(* Logix 5000 project; controller AMANA_DC_PLANT_01 vendor 1 type 14 code 164 rev 31.12; software revision 31.02; part 9 of 9 *)
(* tags used below, declared in another part *)
   Barcode_Longest : DINT;
   Barcode_Shortest : DINT;
   Comma : STRING;
   Counters : COUNTER[16];
   MSG_Enable : DINT;
   MSG_ONS : DINT;
   MSG_Steps : DINT;
   NULL_String : STRING;
   SCANNER_DOCKSORTING_DATA : Keyence_2_Barcode;
   Timer_MSG_Interval : TIMER;
   Read_From_Clearpack_1 : MESSAGE;
   Read_From_L4_1 : MESSAGE;
   Read_From_L6_1 : MESSAGE;
   Read_From_L7_1 : MESSAGE;
   Read_From_Merge_1 : MESSAGE;
   Read_From_Sort_1 : MESSAGE;
(* OH_BARCODE_SCAN, continued *)

ROUTINE R11_DOCKSORTING   (* ladder *)
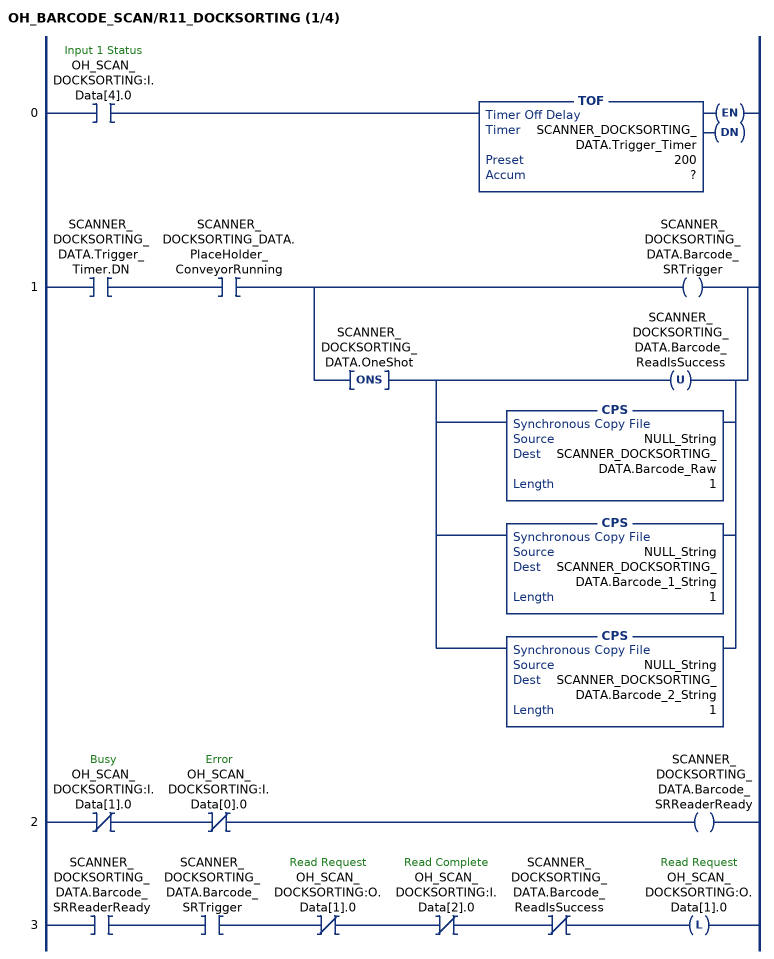
   0: XIC(OH_SCAN_DOCKSORTING:I.Data[4].0)TOF(SCANNER_DOCKSORTING_DATA.Trigger_Timer,?,?);
   1: XIC(SCANNER_DOCKSORTING_DATA.Trigger_Timer.DN)XIC(SCANNER_DOCKSORTING_DATA.PlaceHolder_ConveyorRunning)[OTE(SCANNER_DOCKSORTING_DATA.Barcode_SRTrigger) ,ONS(SCANNER_DOCKSORTING_DATA.OneShot) [OTU(SCANNER_DOCKSORTING_DATA.Barcode_ReadIsSuccess) ,CPS(NULL_String,SCANNER_DOCKSORTING_DATA.Barcode_Raw,1) ,CPS(NULL_String,SCANNER_DOCKSORTING_DATA.Barcode_1_String,1) ,CPS(NULL_String,SCANNER_DOCKSORTING_DATA.Barcode_2_String,1) ] ];
   2: XIO(OH_SCAN_DOCKSORTING:I.Data[1].0)XIO(OH_SCAN_DOCKSORTING:I.Data[0].0)OTE(SCANNER_DOCKSORTING_DATA.Barcode_SRReaderReady);
   3: XIC(SCANNER_DOCKSORTING_DATA.Barcode_SRReaderReady)XIC(SCANNER_DOCKSORTING_DATA.Barcode_SRTrigger)XIO(OH_SCAN_DOCKSORTING:O.Data[1].0)XIO(OH_SCAN_DOCKSORTING:I.Data[2].0)XIO(SCANNER_DOCKSORTING_DATA.Barcode_ReadIsSuccess)OTL(OH_SCAN_DOCKSORTING:O.Data[1].0);
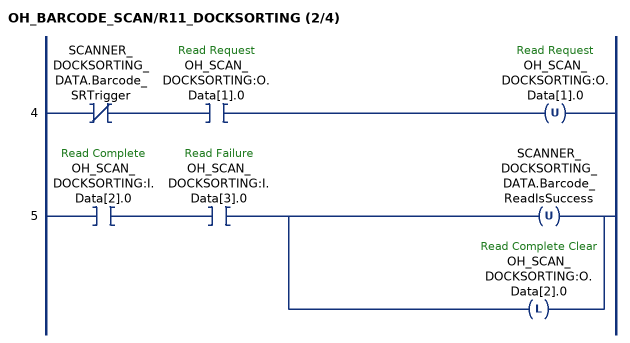
   4: XIO(SCANNER_DOCKSORTING_DATA.Barcode_SRTrigger)XIC(OH_SCAN_DOCKSORTING:O.Data[1].0)OTU(OH_SCAN_DOCKSORTING:O.Data[1].0);
   5: XIC(OH_SCAN_DOCKSORTING:I.Data[2].0)XIC(OH_SCAN_DOCKSORTING:I.Data[3].0)[OTU(SCANNER_DOCKSORTING_DATA.Barcode_ReadIsSuccess) ,OTL(OH_SCAN_DOCKSORTING:O.Data[2].0) ];
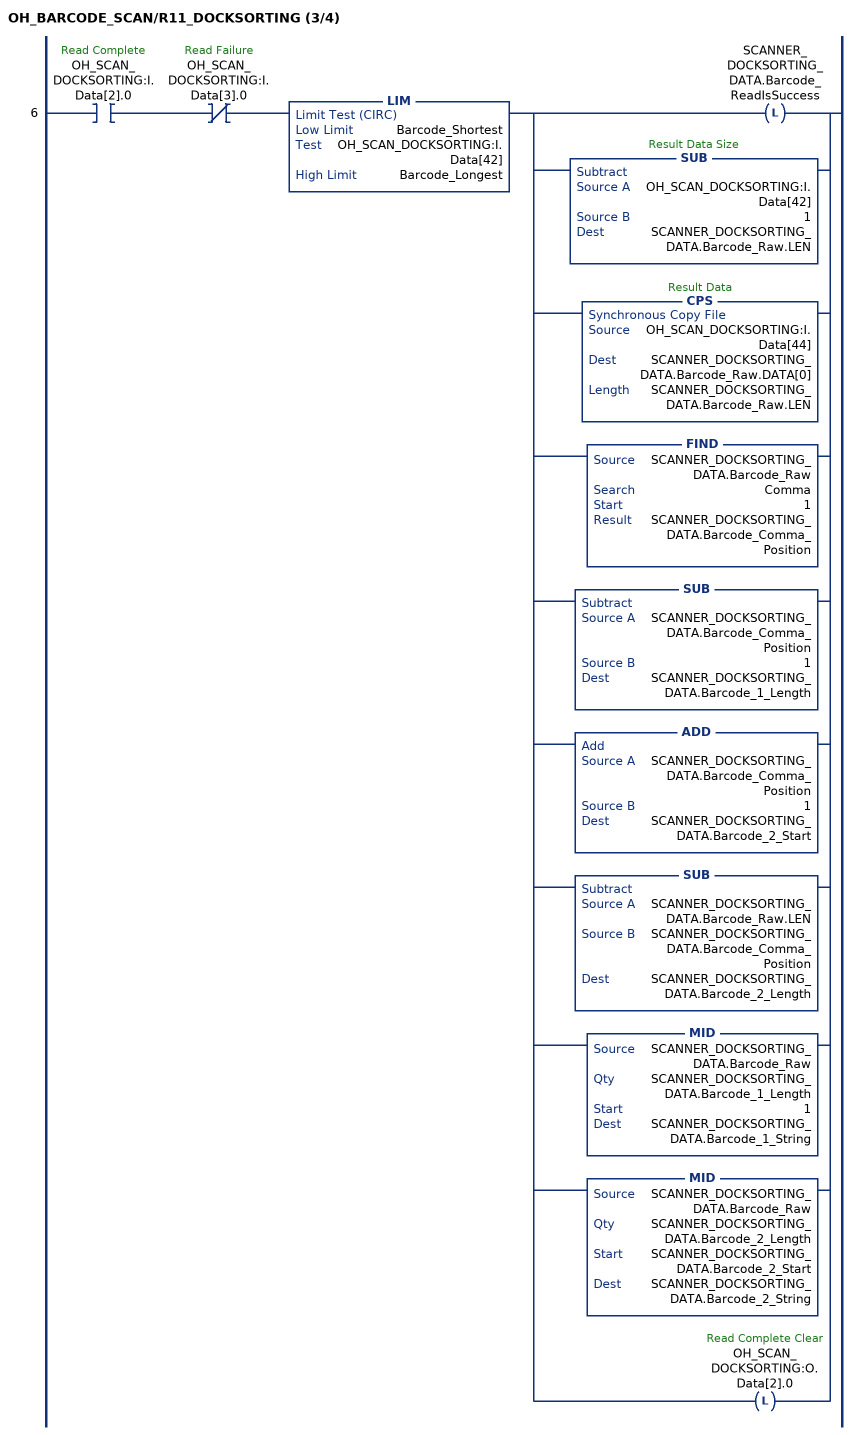
   6: XIC(OH_SCAN_DOCKSORTING:I.Data[2].0)XIO(OH_SCAN_DOCKSORTING:I.Data[3].0)LIM(Barcode_Shortest,OH_SCAN_DOCKSORTING:I.Data[42],Barcode_Longest)[OTL(SCANNER_DOCKSORTING_DATA.Barcode_ReadIsSuccess) ,SUB(OH_SCAN_DOCKSORTING:I.Data[42],1,SCANNER_DOCKSORTING_DATA.Barcode_Raw.LEN) ,CPS(OH_SCAN_DOCKSORTING:I.Data[44],SCANNER_DOCKSORTING_DATA.Barcode_Raw.DATA[0],SCANNER_DOCKSORTING_DATA.Barcode_Raw.LEN) ,FIND(SCANNER_DOCKSORTING_DATA.Barcode_Raw,Comma,1,SCANNER_DOCKSORTING_DATA.Barcode_Comma_Position) ,SUB(SCANNER_DOCKSORTING_DATA.Barcode_Comma_Position,1,SCANNER_DOCKSORTING_DATA.Barcode_1_Length) ,ADD(SCANNER_DOCKSORTING_DATA.Barcode_Comma_Position,1,SCANNER_DOCKSORTING_DATA.Barcode_2_Start) ,SUB(SCANNER_DOCKSORTING_DATA.Barcode_Raw.LEN,SCANNER_DOCKSORTING_DATA.Barcode_Comma_Position,SCANNER_DOCKSORTING_DATA.Barcode_2_Length) ,MID(SCANNER_DOCKSORTING_DATA.Barcode_Raw,SCANNER_DOCKSORTING_DATA.Barcode_1_Length,1,SCANNER_DOCKSORTING_DATA.Barcode_1_String) ,MID(SCANNER_DOCKSORTING_DATA.Barcode_Raw,SCANNER_DOCKSORTING_DATA.Barcode_2_Length,SCANNER_DOCKSORTING_DATA.Barcode_2_Start,SCANNER_DOCKSORTING_DATA.Barcode_2_String) ,OTL(OH_SCAN_DOCKSORTING:O.Data[2].0) ];
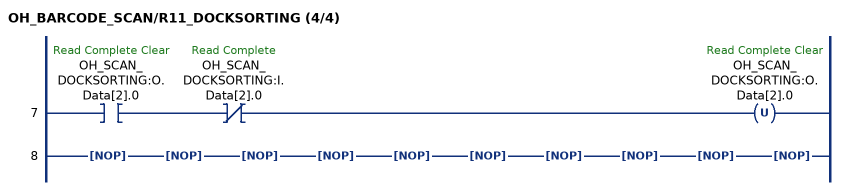
   7: XIC(OH_SCAN_DOCKSORTING:O.Data[2].0)XIO(OH_SCAN_DOCKSORTING:I.Data[2].0)OTU(OH_SCAN_DOCKSORTING:O.Data[2].0);
   8: NOP()NOP()NOP()NOP()NOP()NOP()NOP()NOP()NOP()NOP();
END_ROUTINE

ROUTINE R99_MSG   (* ladder *)
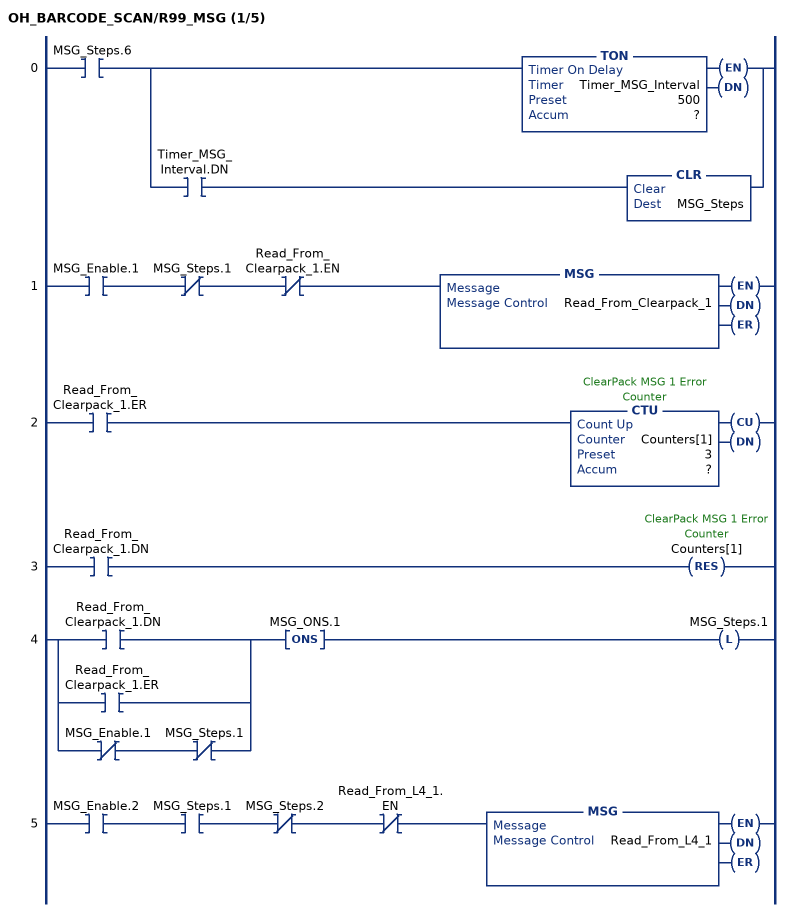
   0: XIC(MSG_Steps.6)[TON(Timer_MSG_Interval,?,?) ,XIC(Timer_MSG_Interval.DN) CLR(MSG_Steps) ];
   1: XIC(MSG_Enable.1)XIO(MSG_Steps.1)XIO(Read_From_Clearpack_1.EN)MSG(Read_From_Clearpack_1);
   2: XIC(Read_From_Clearpack_1.ER)CTU(Counters[1],?,?);
   3: XIC(Read_From_Clearpack_1.DN)RES(Counters[1]);
   4: [XIC(Read_From_Clearpack_1.DN) ,XIC(Read_From_Clearpack_1.ER) ,XIO(MSG_Enable.1) XIO(MSG_Steps.1) ]ONS(MSG_ONS.1)OTL(MSG_Steps.1);
   5: XIC(MSG_Enable.2)XIC(MSG_Steps.1)XIO(MSG_Steps.2)XIO(Read_From_L4_1.EN)MSG(Read_From_L4_1);
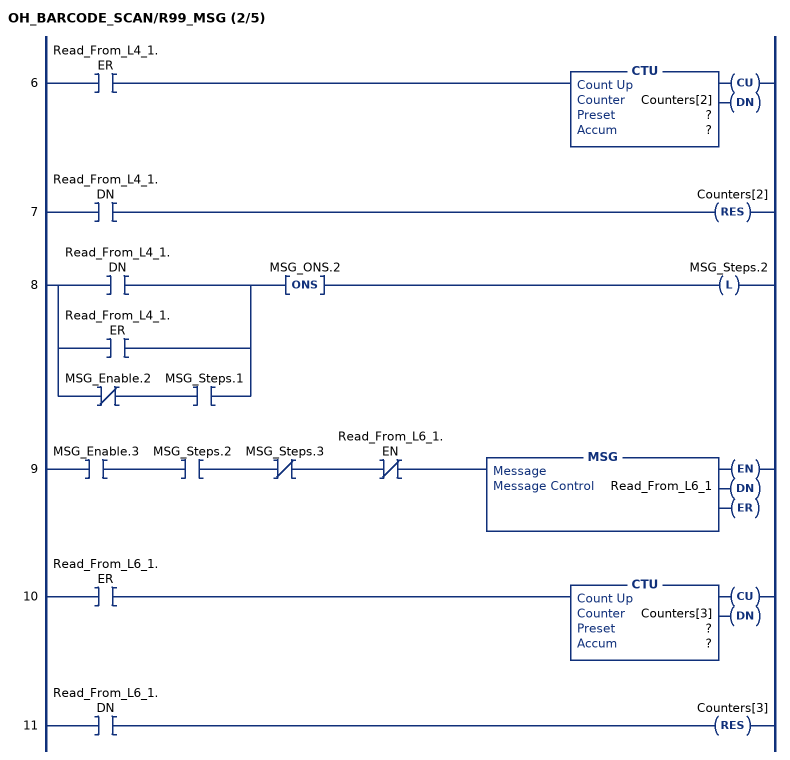
   6: XIC(Read_From_L4_1.ER)CTU(Counters[2],?,?);
   7: XIC(Read_From_L4_1.DN)RES(Counters[2]);
   8: [XIC(Read_From_L4_1.DN) ,XIC(Read_From_L4_1.ER) ,XIO(MSG_Enable.2) XIC(MSG_Steps.1) ]ONS(MSG_ONS.2)OTL(MSG_Steps.2);
   9: XIC(MSG_Enable.3)XIC(MSG_Steps.2)XIO(MSG_Steps.3)XIO(Read_From_L6_1.EN)MSG(Read_From_L6_1);
   10: XIC(Read_From_L6_1.ER)CTU(Counters[3],?,?);
   11: XIC(Read_From_L6_1.DN)RES(Counters[3]);
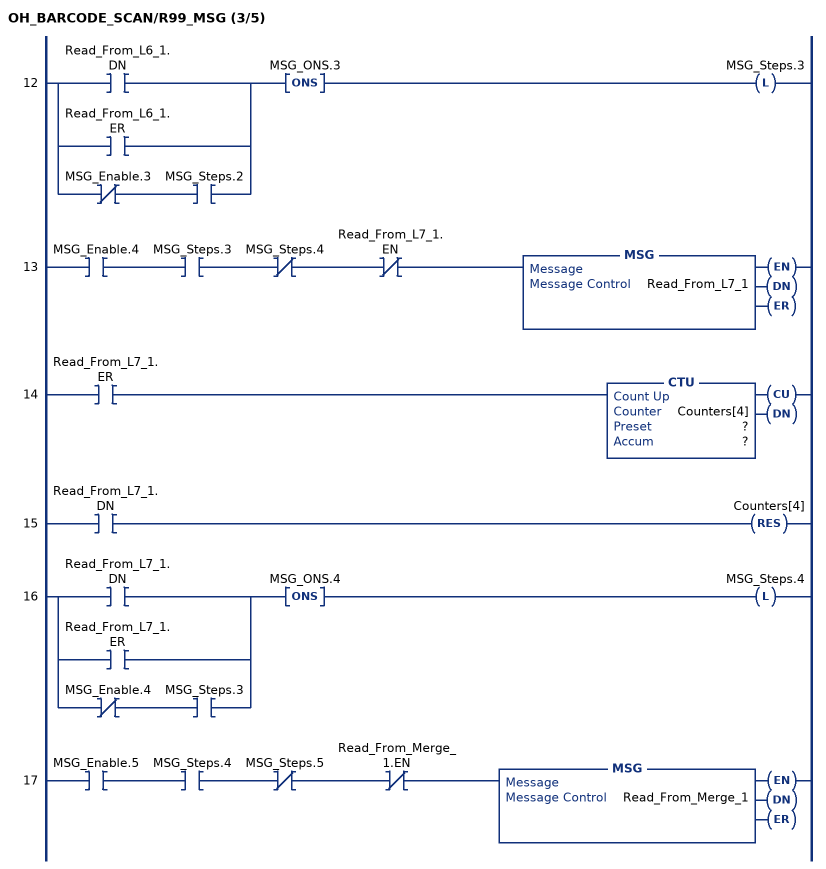
   12: [XIC(Read_From_L6_1.DN) ,XIC(Read_From_L6_1.ER) ,XIO(MSG_Enable.3) XIC(MSG_Steps.2) ]ONS(MSG_ONS.3)OTL(MSG_Steps.3);
   13: XIC(MSG_Enable.4)XIC(MSG_Steps.3)XIO(MSG_Steps.4)XIO(Read_From_L7_1.EN)MSG(Read_From_L7_1);
   14: XIC(Read_From_L7_1.ER)CTU(Counters[4],?,?);
   15: XIC(Read_From_L7_1.DN)RES(Counters[4]);
   16: [XIC(Read_From_L7_1.DN) ,XIC(Read_From_L7_1.ER) ,XIO(MSG_Enable.4) XIC(MSG_Steps.3) ]ONS(MSG_ONS.4)OTL(MSG_Steps.4);
   17: XIC(MSG_Enable.5)XIC(MSG_Steps.4)XIO(MSG_Steps.5)XIO(Read_From_Merge_1.EN)MSG(Read_From_Merge_1);
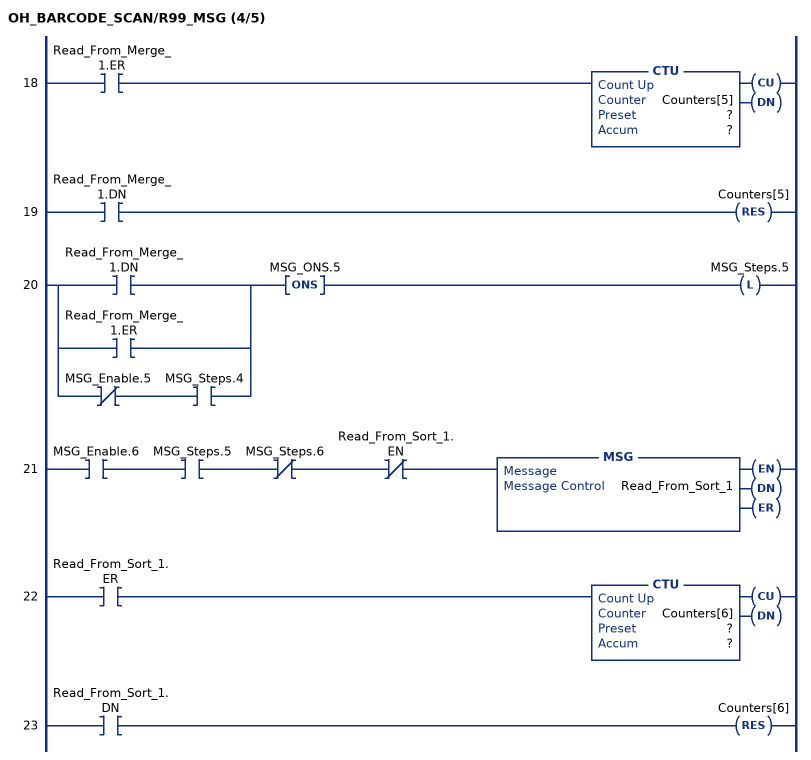
   18: XIC(Read_From_Merge_1.ER)CTU(Counters[5],?,?);
   19: XIC(Read_From_Merge_1.DN)RES(Counters[5]);
   20: [XIC(Read_From_Merge_1.DN) ,XIC(Read_From_Merge_1.ER) ,XIO(MSG_Enable.5) XIC(MSG_Steps.4) ]ONS(MSG_ONS.5)OTL(MSG_Steps.5);
   21: XIC(MSG_Enable.6)XIC(MSG_Steps.5)XIO(MSG_Steps.6)XIO(Read_From_Sort_1.EN)MSG(Read_From_Sort_1);
   22: XIC(Read_From_Sort_1.ER)CTU(Counters[6],?,?);
   23: XIC(Read_From_Sort_1.DN)RES(Counters[6]);
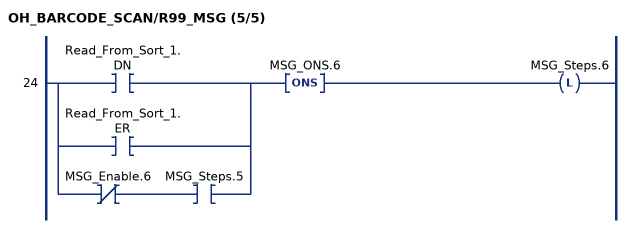
   24: [XIC(Read_From_Sort_1.DN) ,XIC(Read_From_Sort_1.ER) ,XIO(MSG_Enable.6) XIC(MSG_Steps.5) ]ONS(MSG_ONS.6)OTL(MSG_Steps.6);
END_ROUTINE
END_PROGRAM
